TYPE DriveControl :
STRUCT
	Enable : BOOL;
	Reset : BOOL;
END_STRUCT
END_TYPE

(* stored: Version 1.1.0.1, ProductVersion 3.1.4024.11
   DUT DriveControl: Id {f3c58783-e1ab-4de7-9ca0-889574d965d2} *)
